(* IEC 61131-3 sources: OT-Lab/scripts/v2_seed, 1 file *)

(* ---- openplc_bool_minimal.st ---- *)
PROGRAM plc_prg
VAR
    SWITCH_CMD AT %QX0.0 : BOOL;
END_VAR

END_PROGRAM

CONFIGURATION Config0
    RESOURCE Res0 ON PLC
        TASK Main(INTERVAL := T#100ms, PRIORITY := 0);
        PROGRAM Inst0 WITH Main : plc_prg;
    END_RESOURCE
END_CONFIGURATION
